FUNCTION_BLOCK FB_SystemCalibrationTestDouble IMPLEMENTS I_SystemCalibration
VAR
    bIsCalibrated : BOOL;
END_VAR


METHOD IsCalibrated : BOOL
IsCalibrated := THIS^.bIsCalibrated;
END_METHOD

METHOD SetIsCalibrated : BOOL
VAR_INPUT
    bIsCalibrated : BOOL;
END_VAR
THIS^.bIsCalibrated := bIsCalibrated;
END_METHOD

END_FUNCTION_BLOCK

(* stored: Version 1.1.0.1
   POU FB_SystemCalibrationTestDouble: Id {c489bb26-745f-45fc-b640-3153c052ad06}, SpecialFunc None
   Method IsCalibrated: Id {d983f7d3-9c09-47aa-a8e0-cd048dd8a7cc}
   Method SetIsCalibrated: Id {8e69450e-2e7b-408c-bfd8-ad3d41c2a492} *)
